INTERFACE ITcoMultiAxis

METHOD MoveAbsolute : TcoCore.ITcoTaskStatus
VAR_INPUT
	MoveParams : TcoMultiAxisMoveParam;;
END_VAR
END_METHOD

PROPERTY MoveAbsoluteTask : REFERENCE TO TcoCore.TcoTask
GET
END_GET
END_PROPERTY

METHOD ResetDrives : TcoCore.ITcoTaskStatus
VAR_INPUT
END_VAR
END_METHOD

METHOD SoeReset : TcoCore.ITcoTaskStatus
VAR_INPUT
END_VAR
END_METHOD

END_INTERFACE

(* stored: Version 1.1.0.1, ProductVersion 3.1.4024.12
   Itf ITcoMultiAxis: Id {2806ae3f-4ed0-01df-236d-2a72bef75673}
   Method MoveAbsolute: Id {3d93c280-34a3-0858-3005-13005fbeb679}
   Property MoveAbsoluteTask: Id {eab7a3c0-bbcf-0162-2b43-cb974293fed7}
   Get Get: Id {eed0ea8e-ad14-0093-1a66-95b402c0db4d}
   Method ResetDrives: Id {7f0de09b-71f1-0d98-362c-975550baa88c}
   Method SoeReset: Id {f4881921-cdf0-0d8c-32a5-0fec87c316d9} *)
